// SIMATIC S7-200 project (STEP 7-Micro/WIN), CPU 226 REL 02.00

SYMBOL_TABLE 用户定义1
状态               M0.0     // 程序执行的状态，是否完成操作。正在操作时为1。
current_x        MD20     // 当前所处的x坐标
current_y        MD24     // 当前所处的y坐标
仓库号              MW28     // 所选的仓库号
count_time       MW10     // 脉冲发生定时器的数值
K8入库             M0.1
K12出库            M0.2
按键号              VW238    // 当前的按键号
END_SYMBOL_TABLE

SYMBOL_TABLE S7-200 符号
Always_On        SM0.0    // 始终接通为 ON
First_Scan_On    SM0.1    // 仅第一个扫描周期中接通为 ON
PLS0_Idle        SM66.7   // PTO0 空闲：0 = PTO 正在执行；1 = PTO 空闲
PLS1_Idle        SM76.7   // PTO1 空闲：0 = PTO正在执行；1 = PTO空闲
PLS0_Ctrl        SMB67    // PTO0/PMW0 监控，用于 Q0.0 上的 PTO（脉冲串输出）和PWM（脉冲宽度调制）
PTO0_PC          SMD72    // PTO0 脉冲计数值：双字整数（1至2^32 - 1）
PLS0_Cycle       SMW68    // PTO0/PWM0 周期时间值：字数据类型（2 至 65,535 个时基单位）
PTO0_Profile     SMW168   // PTO0 包络表的 V 存储区起始地址（对 V0 的偏移量，字数据类型）
END_SYMBOL_TABLE

ORGANIZATION_BLOCK 主程序:OB1
TITLE=立体仓库控制
BEGIN
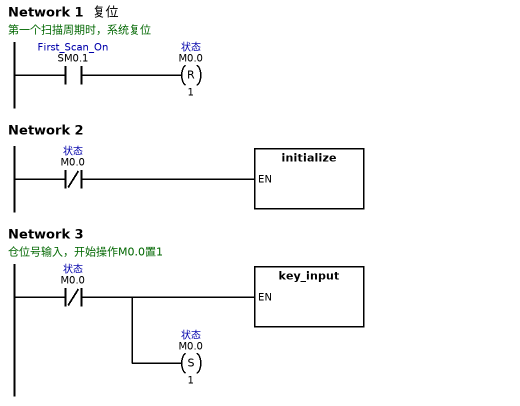
Network 1 // 复位
// 第一个扫描周期时，系统复位
LD     First_Scan_On:SM0.1
R      状态:M0.0, 1
Network 2
LDN    状态:M0.0
CALL   initialize:SBR0
Network 3
// 仓位号输入，开始操作M0.0置1
LDN    状态:M0.0
CALL   key_input:SBR4
S      状态:M0.0, 1
END_ORGANIZATION_BLOCK

SUBROUTINE_BLOCK initialize:SBR0
TITLE=初始化
BEGIN
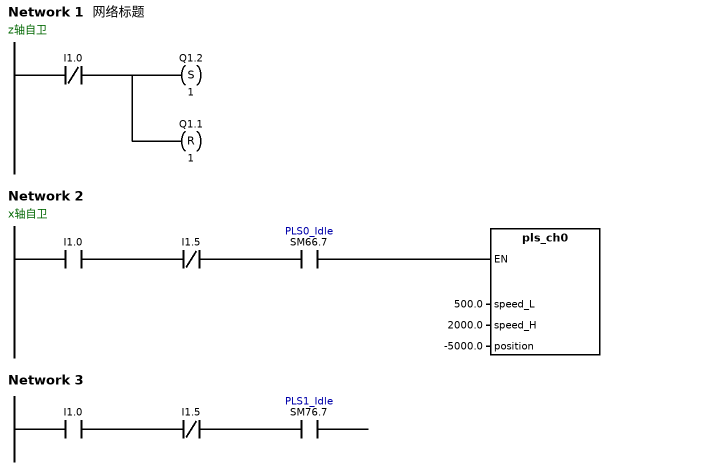
Network 1 // 网络标题
// z轴自卫
LDN    I1.0
S      Q1.2, 1
R      Q1.1, 1
Network 2
// x轴自卫 
LD     I1.0
AN     I1.5
A      PLS0_Idle:SM66.7
CALL   pls_ch0:SBR1, 500.0, 2000.0, -5000.0
Network 3
// (network saved uncompiled; LAD cells follow)
// row 0: c0 -| |- I1.0  c1 -|/|- I1.5  c2 -| |- PLS1_Idle:SM76.7
END_SUBROUTINE_BLOCK

SUBROUTINE_BLOCK pls_ch0:SBR1
TITLE=脉冲发生器0的控制程序 x轴
VAR_INPUT
speed_L:REAL;	// LD0 起始速度
speed_H:REAL;	// LD4 运行速度
position:REAL;	// LD8 目标位置（绝对坐标，系统即将到达的目标脉冲数）
END_VAR
BEGIN
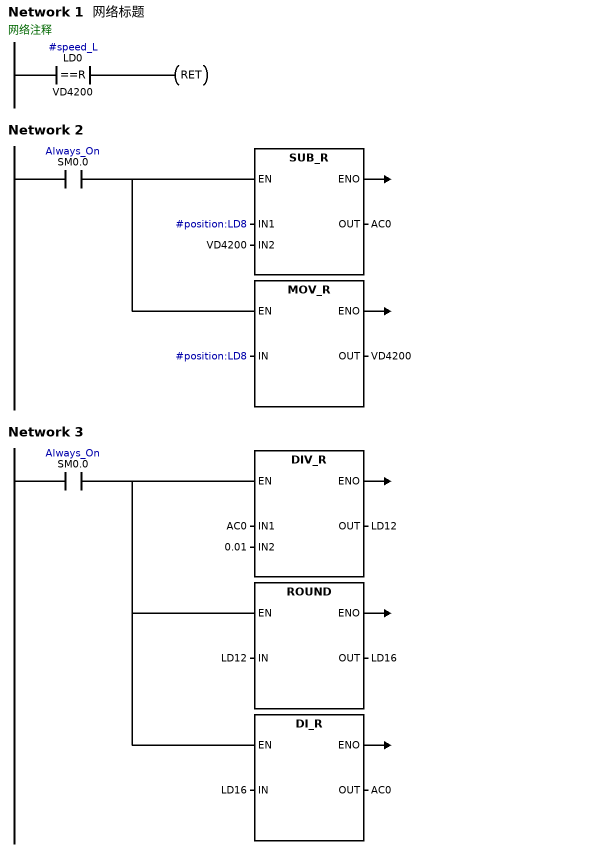
Network 1 // 网络标题
// 网络注释
LDR=   #speed_L:LD0, VD4200
CRET
Network 2
LD     Always_On:SM0.0
MOVR   #position:LD8, AC0
-R     VD4200, AC0
MOVR   #position:LD8, VD4200
Network 3
LD     Always_On:SM0.0
MOVR   AC0, LD12
/R     0.01, LD12
ROUND  LD12, LD16
DTR    LD16, AC0
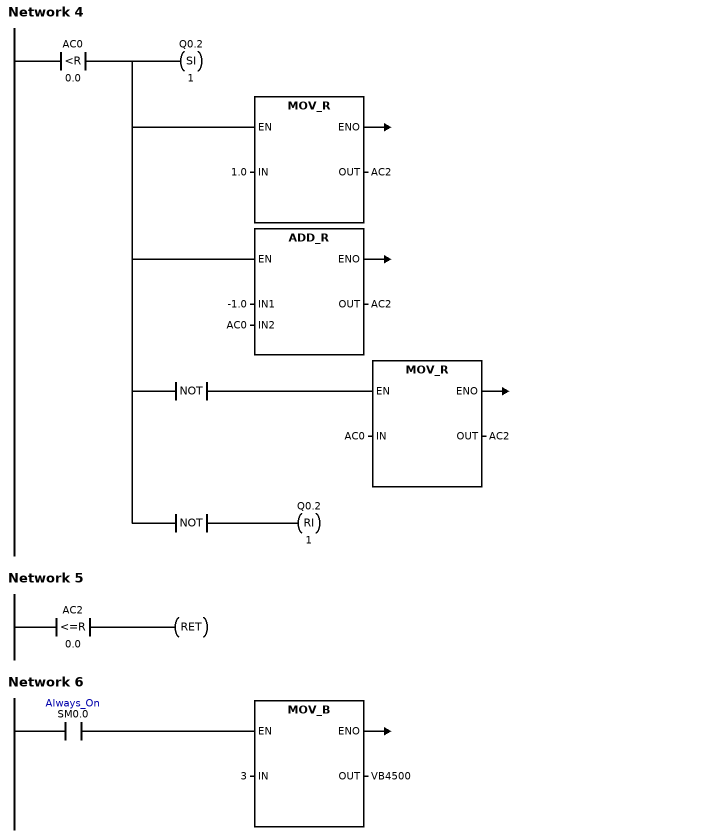
Network 4
LDR<   AC0, 0.0
LPS
SI     Q0.2, 1
MOVR   1.0, AC2
MOVR   -1.0, AC2
+R     AC0, AC2
NOT
MOVR   AC0, AC2
LPP
NOT
RI     Q0.2, 1
Network 5
LDR<=  AC2, 0.0
CRET
Network 6
LD     Always_On:SM0.0
MOVB   3, VB4500
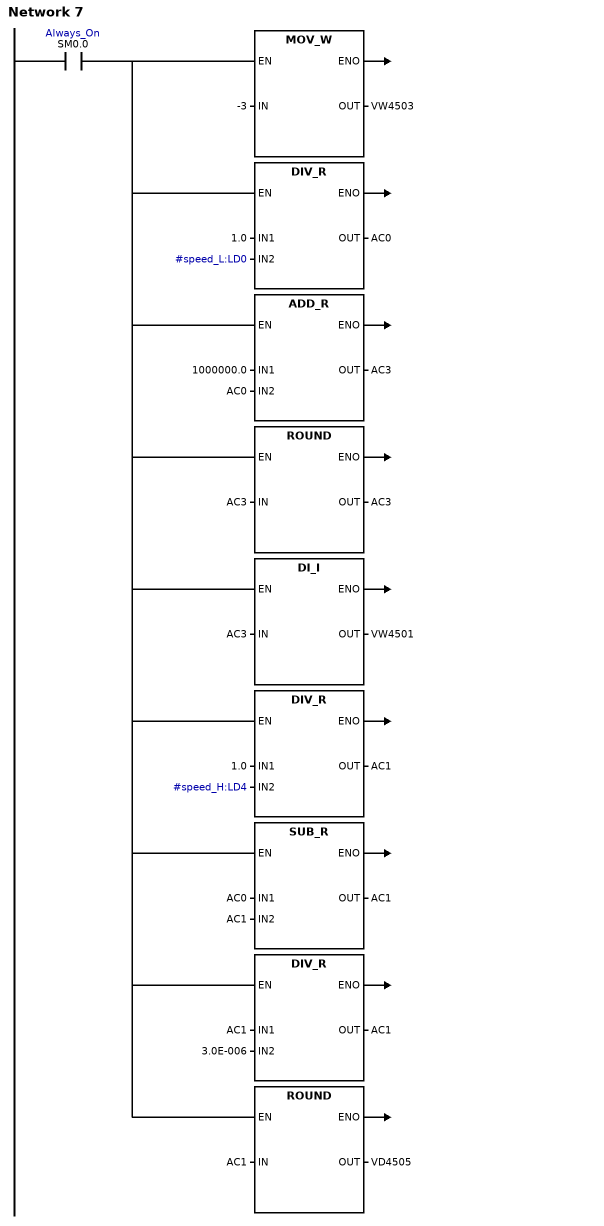
Network 7
LD     Always_On:SM0.0
MOVW   -3, VW4503
MOVR   1.0, AC0
/R     #speed_L:LD0, AC0
MOVR   1000000.0, AC3
+R     AC0, AC3
ROUND  AC3, AC3
DTI    AC3, VW4501
MOVR   1.0, AC1
/R     #speed_H:LD4, AC1
*R     -1.0, AC1
+R     AC0, AC1
/R     3.0E-006, AC1
ROUND  AC1, VD4505
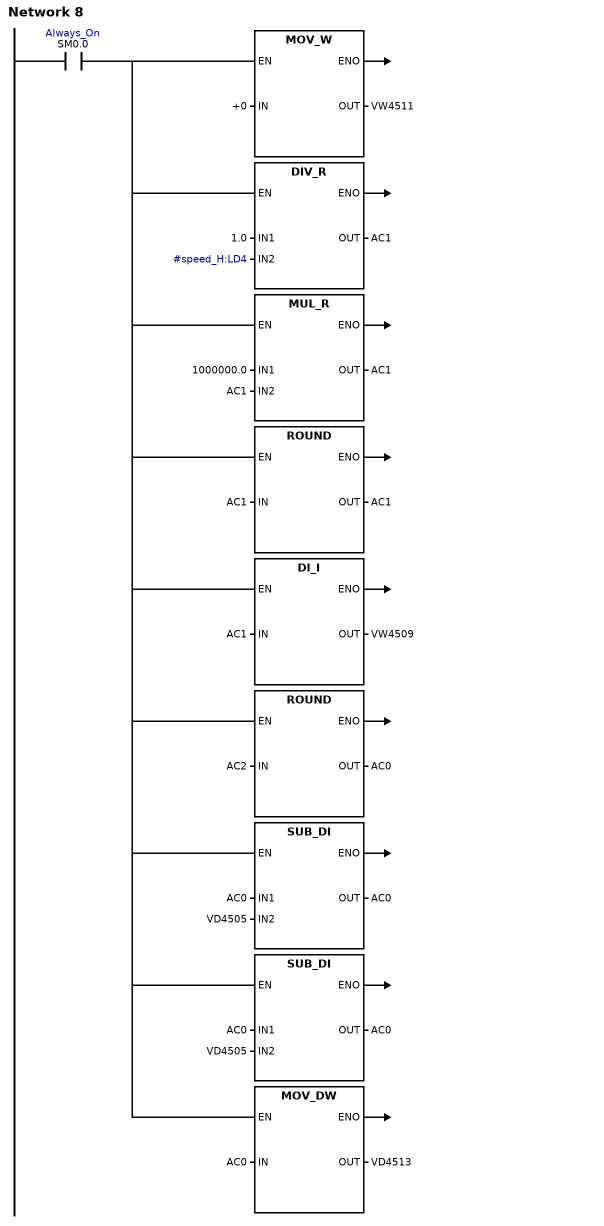
Network 8
LD     Always_On:SM0.0
MOVW   +0, VW4511
MOVR   1.0, AC1
/R     #speed_H:LD4, AC1
*R     1000000.0, AC1
ROUND  AC1, AC1
DTI    AC1, VW4509
ROUND  AC2, AC0
-D     VD4505, AC0
-D     VD4505, AC0
MOVD   AC0, VD4513
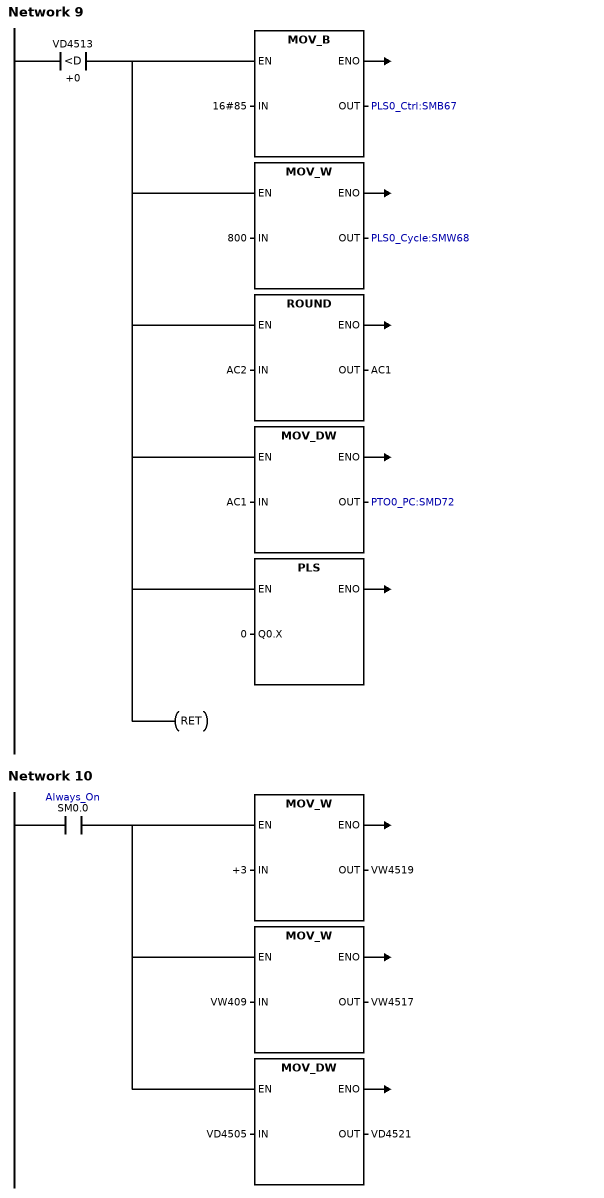
Network 9
LDD<   VD4513, +0
MOVB   16#85, PLS0_Ctrl:SMB67
MOVW   800, PLS0_Cycle:SMW68
ROUND  AC2, AC1
MOVD   AC1, PTO0_PC:SMD72
PLS    0
CRET
Network 10
LD     Always_On:SM0.0
MOVW   +3, VW4519
MOVW   VW409, VW4517
MOVD   VD4505, VD4521
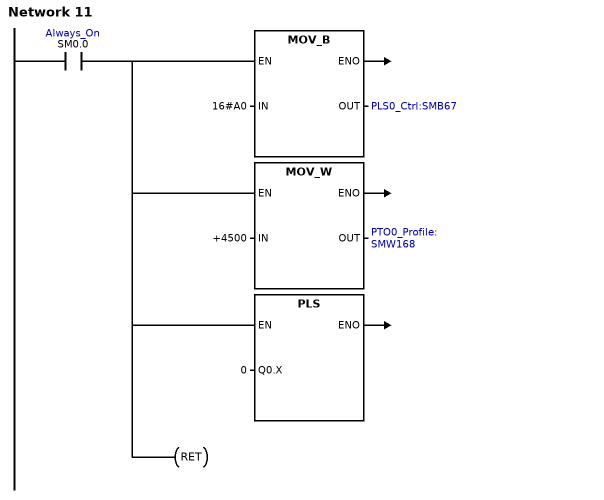
Network 11
LD     Always_On:SM0.0
MOVB   16#A0, PLS0_Ctrl:SMB67
MOVW   +4500, PTO0_Profile:SMW168
PLS    0
CRET
Network 16 // 网络标题
// 网络注释
END_SUBROUTINE_BLOCK

SUBROUTINE_BLOCK pls_ch1:SBR2
TITLE=脉冲发生器1的控制程序 y轴
VAR_INPUT
speed_L:REAL;	// LD0 
speed_H:REAL;	// LD4 
position:REAL;	// LD8 
END_VAR
BEGIN
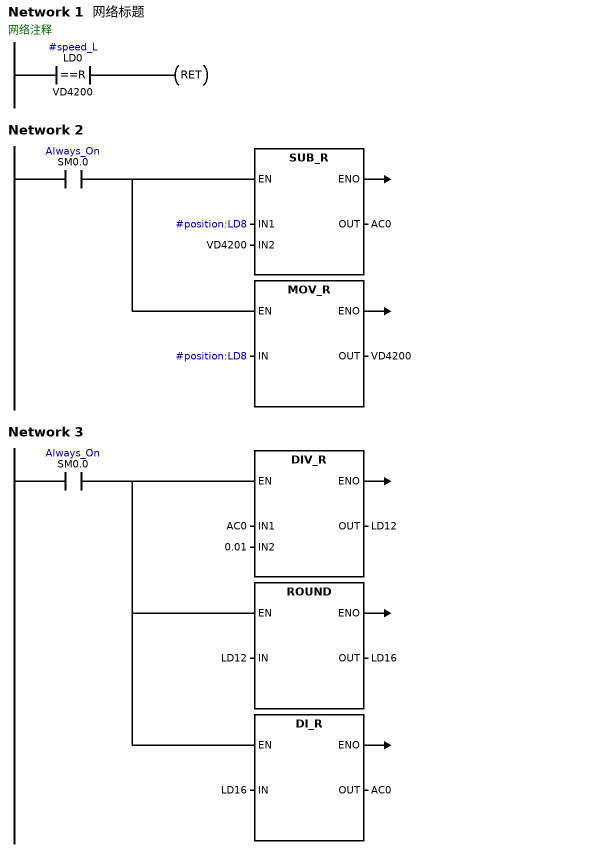
Network 1 // 网络标题
// 网络注释
LDR=   #speed_L:LD0, VD4200
CRET
Network 2
LD     Always_On:SM0.0
MOVR   #position:LD8, AC0
-R     VD4200, AC0
MOVR   #position:LD8, VD4200
Network 3
LD     Always_On:SM0.0
MOVR   AC0, LD12
/R     0.01, LD12
ROUND  LD12, LD16
DTR    LD16, AC0
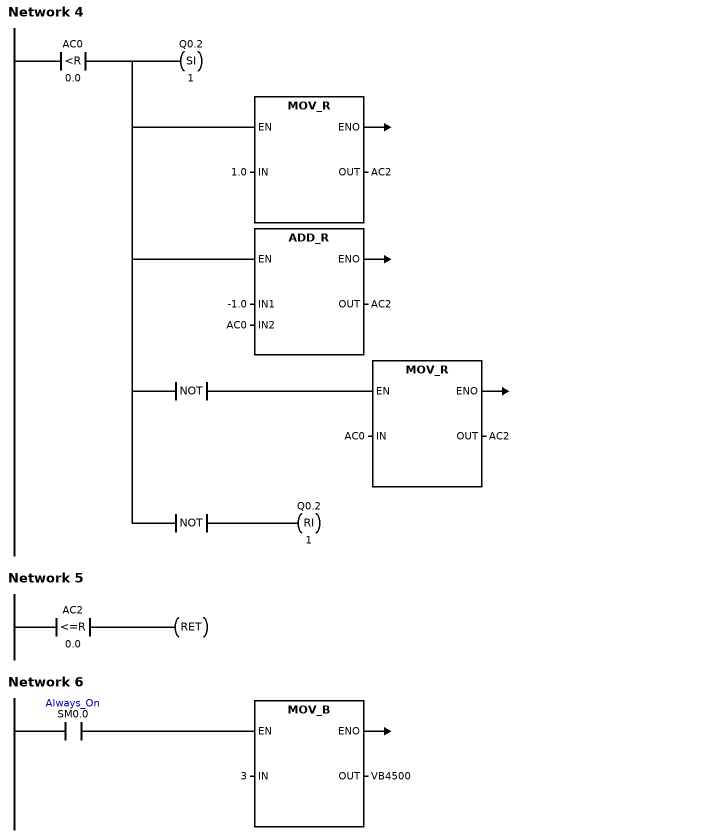
Network 4
LDR<   AC0, 0.0
LPS
SI     Q0.2, 1
MOVR   1.0, AC2
MOVR   -1.0, AC2
+R     AC0, AC2
NOT
MOVR   AC0, AC2
LPP
NOT
RI     Q0.2, 1
Network 5
LDR<=  AC2, 0.0
CRET
Network 6
LD     Always_On:SM0.0
MOVB   3, VB4500
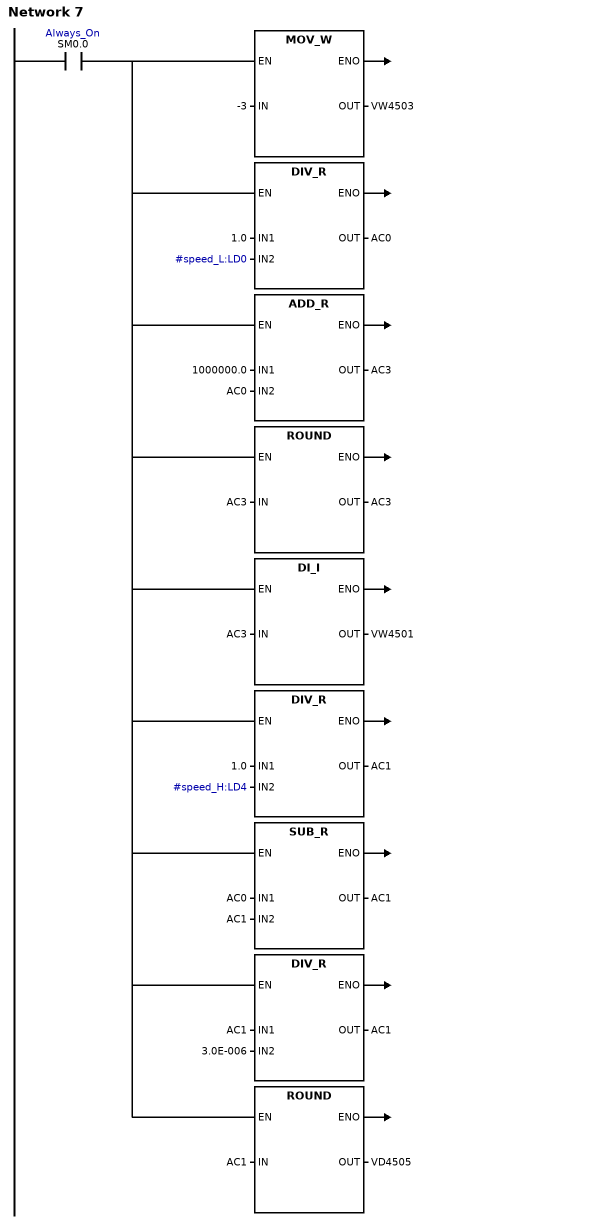
Network 7
LD     Always_On:SM0.0
MOVW   -3, VW4503
MOVR   1.0, AC0
/R     #speed_L:LD0, AC0
MOVR   1000000.0, AC3
+R     AC0, AC3
ROUND  AC3, AC3
DTI    AC3, VW4501
MOVR   1.0, AC1
/R     #speed_H:LD4, AC1
*R     -1.0, AC1
+R     AC0, AC1
/R     3.0E-006, AC1
ROUND  AC1, VD4505
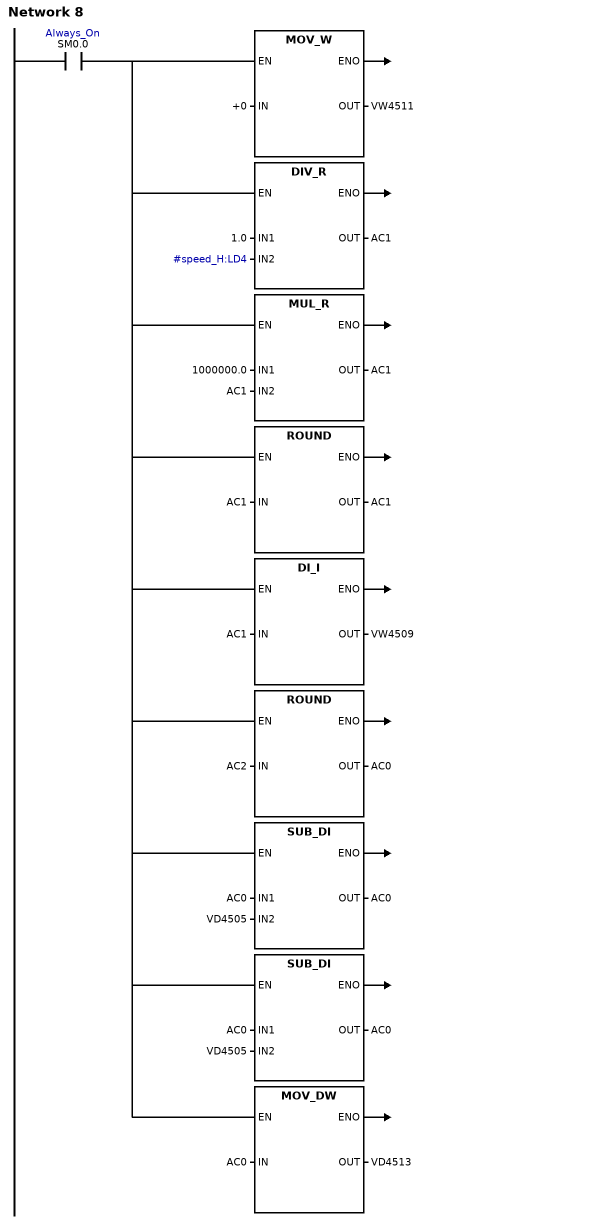
Network 8
LD     Always_On:SM0.0
MOVW   +0, VW4511
MOVR   1.0, AC1
/R     #speed_H:LD4, AC1
*R     1000000.0, AC1
ROUND  AC1, AC1
DTI    AC1, VW4509
ROUND  AC2, AC0
-D     VD4505, AC0
-D     VD4505, AC0
MOVD   AC0, VD4513
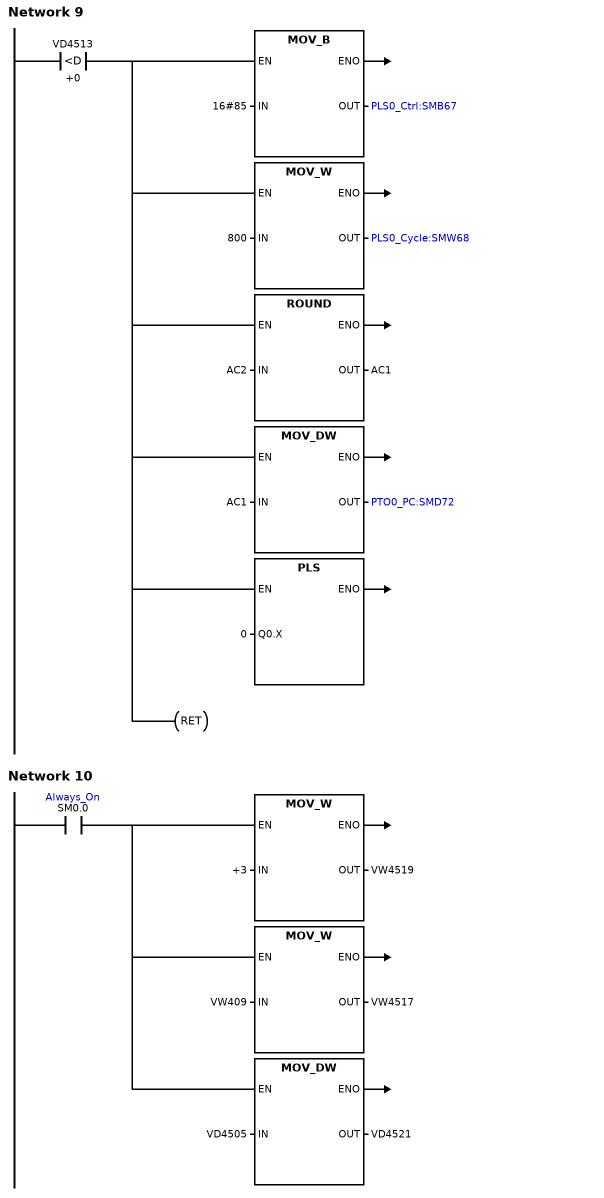
Network 9
LDD<   VD4513, +0
MOVB   16#85, PLS0_Ctrl:SMB67
MOVW   800, PLS0_Cycle:SMW68
ROUND  AC2, AC1
MOVD   AC1, PTO0_PC:SMD72
PLS    0
CRET
Network 10
LD     Always_On:SM0.0
MOVW   +3, VW4519
MOVW   VW409, VW4517
MOVD   VD4505, VD4521
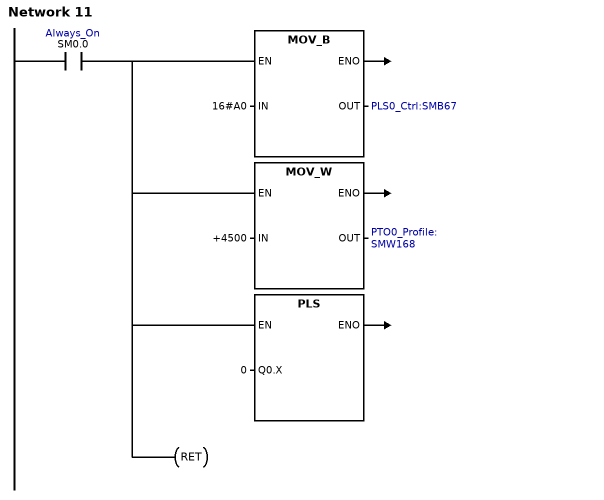
Network 11
LD     Always_On:SM0.0
MOVB   16#A0, PLS0_Ctrl:SMB67
MOVW   +4500, PTO0_Profile:SMW168
PLS    0
CRET
Network 16 // 网络标题
// 网络注释
Network 26 // 网络标题
// 网络注释
END_SUBROUTINE_BLOCK

SUBROUTINE_BLOCK scan:SBR3
TITLE=键盘扫描程序
BEGIN
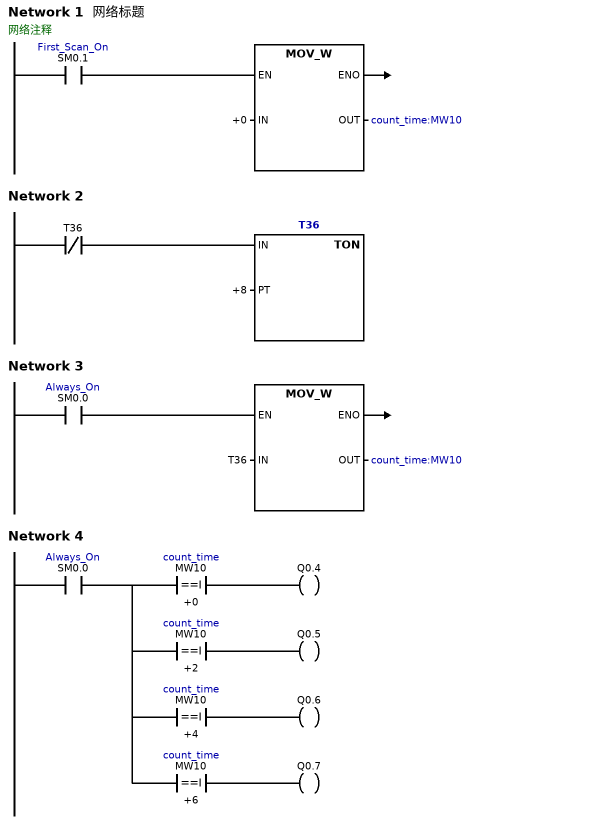
Network 1 // 网络标题
// 网络注释
LD     First_Scan_On:SM0.1
MOVW   +0, count_time:MW10
Network 2
LDN    T36
TON    T36, +8
Network 3
LD     Always_On:SM0.0
MOVW   T36, count_time:MW10
Network 4
LD     Always_On:SM0.0
LPS
AW=    count_time:MW10, +0
=      Q0.4
LRD
AW=    count_time:MW10, +2
=      Q0.5
LRD
AW=    count_time:MW10, +4
=      Q0.6
LPP
AW=    count_time:MW10, +6
=      Q0.7
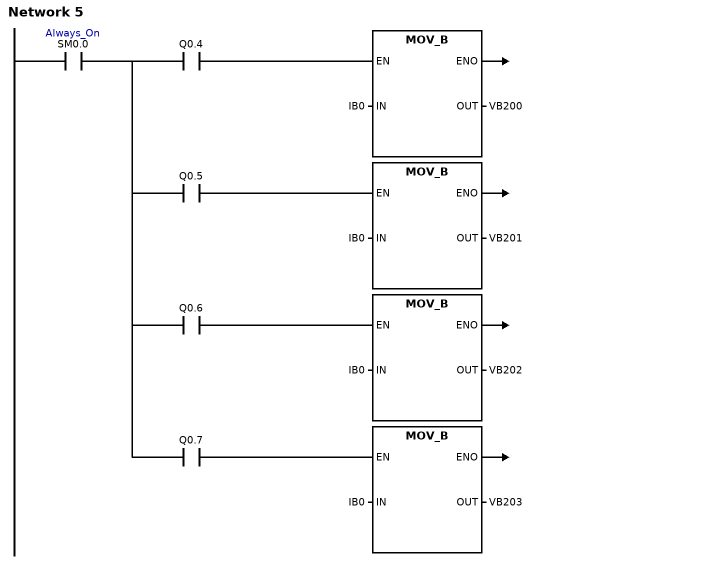
Network 5
LD     Always_On:SM0.0
LPS
A      Q0.4
MOVB   IB0, VB200
LRD
A      Q0.5
MOVB   IB0, VB201
LRD
A      Q0.6
MOVB   IB0, VB202
LPP
A      Q0.7
MOVB   IB0, VB203
Network 11 // 网络标题
// 网络注释
END_SUBROUTINE_BLOCK

SUBROUTINE_BLOCK key_input:SBR4
TITLE=存储键盘输入的值
BEGIN
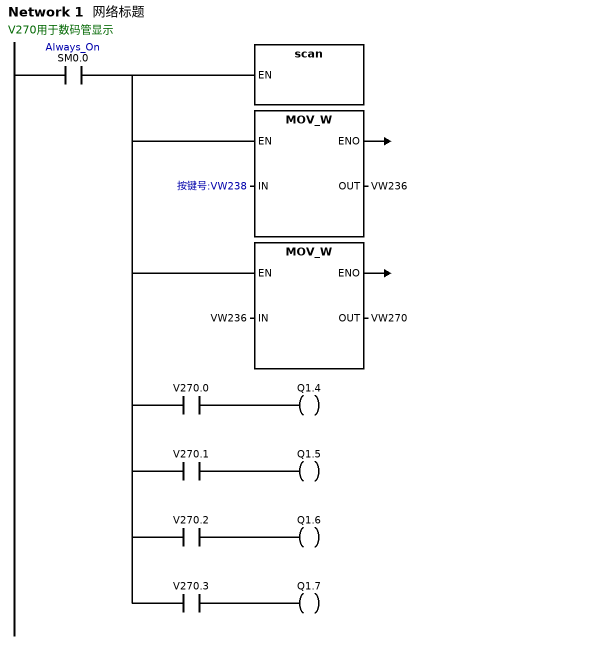
Network 1 // 网络标题
// V270用于数码管显示
LD     Always_On:SM0.0
LPS
CALL   scan:SBR3
MOVW   按键号:VW238, VW236
MOVW   VW236, VW270
A      V270.0
=      Q1.4
LRD
A      V270.1
=      Q1.5
LRD
A      V270.2
=      Q1.6
LPP
A      V270.3
=      Q1.7
Network 2
// 将扫描的结果送入VW240，得到
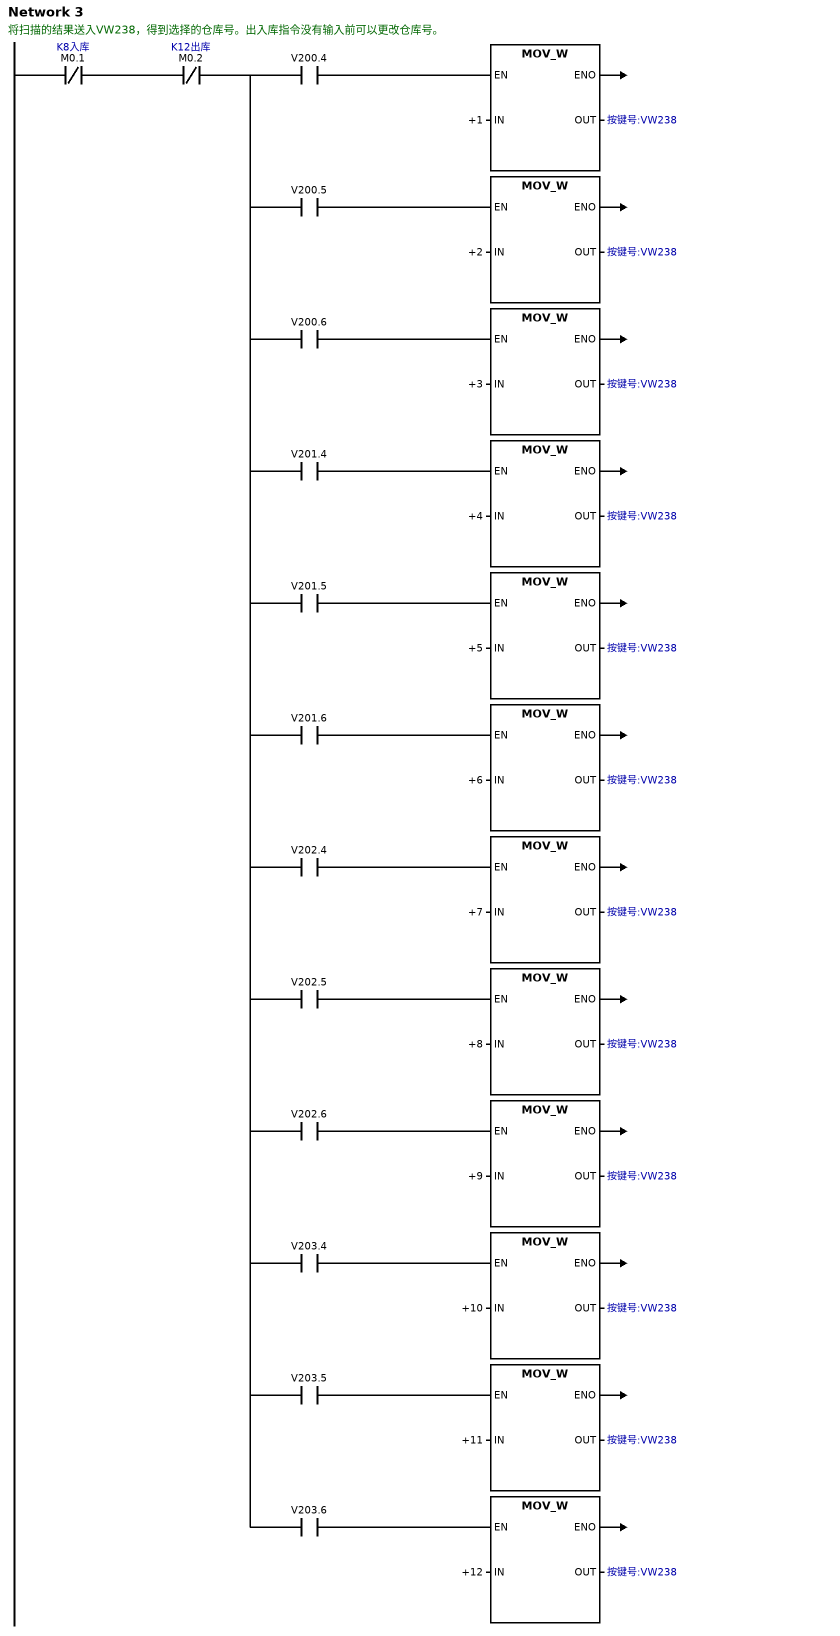
Network 3
// 将扫描的结果送入VW238，得到选择的仓库号。出入库指令没有输入前可以更改仓库号。
LDN    K8入库:M0.1
AN     K12出库:M0.2
LPS
A      V200.4
MOVW   +1, 按键号:VW238
LRD
A      V200.5
MOVW   +2, 按键号:VW238
LRD
A      V200.6
MOVW   +3, 按键号:VW238
LRD
A      V201.4
MOVW   +4, 按键号:VW238
LRD
A      V201.5
MOVW   +5, 按键号:VW238
LRD
A      V201.6
MOVW   +6, 按键号:VW238
LRD
A      V202.4
MOVW   +7, 按键号:VW238
LRD
A      V202.5
MOVW   +8, 按键号:VW238
LRD
A      V202.6
MOVW   +9, 按键号:VW238
LRD
A      V203.4
MOVW   +10, 按键号:VW238
LRD
A      V203.5
MOVW   +11, 按键号:VW238
LPP
A      V203.6
MOVW   +12, 按键号:VW238
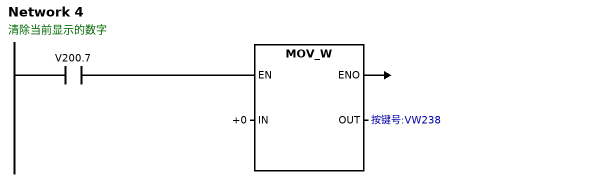
Network 4
// 清除当前显示的数字
LD     V200.7
MOVW   +0, 按键号:VW238
Network 12 // 网络标题
// 网络注释
END_SUBROUTINE_BLOCK
